(* IEC 61131-3 sources: teller/JD_Teller_LC2_V11/Class/CAIInputChannel, 1 file *)

(* ---- CAIInputChannel.st ---- *)
(*!
<Class
	Name               = "CAIInputChannel"
	Revision           = "2.20"
	RealtimeTask       = "false"
	CyclicTask         = "false"
	BackgroundTask     = "false"
	Sigmatek           = "true"
	OSInterface        = "false"
	HighPriority       = "false"
	Automatic          = "false"
	UpdateMode         = "Prescan"
	IconPath           = ".\Class\Tool.ico"
	SharedCommandTable = "true"
	Objectsize         = "(284,120)">
	<Channels>
		<Client Name="connectc" Required="true" Internal="false"/>
		<Client Name="EEOffset" Required="true" Internal="false"/>
		<Client Name="Neg" Required="false" Internal="false"/>
	</Channels>
	<RevDoku>
		<Owner Company="Sigmatek" Author="stewer"/>
		<Dokumentation Revision="2.20" Date="05.12.2013" Author="LanSte&#13;&#10;FucHer" Company="Sigmatek" Description="Added payload support&#13;&#10;Changed AWL code to Structured Text. CyRt Client default value: 1"/>
		<Dokumentation Revision="2.11" Date="04.03.2010" Author="BleErn" Company="Sigmatek" Description="Changes in BaseClass (UpdateRtPostScan)"/>
	</RevDoku>
	<Network Name="CAIInputChannel">
		<!-- List of Components in this network -->
		<Components>
			<Object
				Name       = "_base"
				Class      = "DAIInputChnl"
				Position   = "(270,150)"
				Visualized = "true">
				<Channels>
					<Server Name="Data"/>
					<Server Name="State"/>
					<Client Name="BitResolution"/>
					<Client Name="CBias"/>
					<Client Name="channel"/>
					<Client Name="CInvert"/>
					<Client Name="connect"/>
					<Client Name="CScale"/>
					<Client Name="CyRt" Value="1"/>
					<Client Name="TypeofChannel"/>
				</Channels>
			</Object>
		</Components>
		<Comments>
		</Comments>
		<!-- List of Connections in this network -->
		<Connections>
			<Connection Source="this.Data" Destination="_base.Data" Vertices="(742,210),(570,240),"/>
			<Connection Source="this.State" Destination="_base.State" Vertices="(742,270),(570,300),"/>
			<Connection Source="_base.TypeofChannel" Destination="this.TypeofChannel" Vertices="(270,360),(38,270),"/>
			<Connection Source="_base.CyRt" Destination="this.CyRt" Vertices="(270,420),(38,330),"/>
			<Connection Source="_base.CScale" Destination="this.CScale" Vertices="(270,480),(38,390),"/>
			<Connection Source="_base.CBias" Destination="this.CBias" Vertices="(270,540),(38,450),"/>
			<Connection Source="_base.CInvert" Destination="this.CInvert" Vertices="(270,600),(38,510),"/>
			<Connection Source="_base.BitResolution" Destination="this.BitResolution" Vertices="(270,660),(38,570),"/>
			<Connection Source="_base.channel" Destination="this.channel" Vertices="(270,240),(38,210),"/>
		</Connections>
		<!-- Headerfiles -->
		<Options>
		</Options>
	</Network>
</Class>
*)
#pragma using DAIInputChnl

CAIInputChannel : CLASS
: DAIInputChnl
  //Servers:
  //Clients:
	connectc 	: CltChCmd_HwBaseCDIAS;
	Neg 	: CltCh_DINT;
	EEOffset 	: CltCh_DINT;
  //Variables:
  //Functions:
				//! <Function Comment="[#ENGLISH]&#13;&#10; *******************************************************&#13;&#10; this is the init method of one input channel&#13;&#10; *******************************************************&#13;&#10;" Name="Init"/>
	FUNCTION VIRTUAL GLOBAL Init;

	FUNCTION CalFactory1;
				//! <Function Comment="-- overwite this function if there are other offsets ---------------------------&#13;&#10;" Name="GetEEOffset"/>
	FUNCTION VIRTUAL GLOBAL GetEEOffset
		VAR_OUTPUT
			Offset 	: UINT;
		END_VAR;

	FUNCTION GLOBAL ReCallFactory;

	FUNCTION VIRTUAL GLOBAL SetBalanceData;

	FUNCTION AWL CalFactory1_AWL;
  //Tables:
	FUNCTION @STD
		VAR_OUTPUT
			ret_code	: CONFSTATES;
		END_VAR;
	FUNCTION GLOBAL TAB @CT_;
END_CLASS;

#pragma usingLtd HwBaseCDIAS

#pragma usingLtd DiasMaster

(****************************************************************************************
*
*	Created : Sigmatek
*	Changes :
*		2.5 => 2.10	/	05.12.2007	/	Mark:	//#SR001
*			- [DB 713]: make compatible to CIV/DIV DataMover
*		1.1 => 2.5	/	06.03.2007	/	Mark:	//#SR000
*			- [DB 421]: now class is ready for plug & play over CIV
*		0.1 => 1.1 / 23.12.2004 / no Mark / ws
*			compatibility with Lasal Class 2
*			removed visible flags from internal servers
*
*****************************************************************************************)

//[#ENGLISH]
// *******************************************************
// this is the init method of one input channel
// *******************************************************
FUNCTION VIRTUAL GLOBAL CAIInputChannel::Init

	channel       := channel.read();
	TypeofChannel := TypeofChannel.read();
	CyRt          := CyRt.read();
	CScale        := CScale.read();
	CBias         := CBias.read();
	CInvert 	  := CInvert.read();
	BitResolution := BitResolution.read();
	Neg := Neg.Read();
	EEOffset := EEOffset.Read();

	if BitResolution = 14 then
		udMaxBin := 16000;
	else
		udMaxBin := 4000;
	end_if;

	//#SR000 start
	b_VaranAvailable := Connectc.Masterconnect.IsVaranAvailable() <> 0;

	if ( b_VaranAvailable = TRUE ) then
		if firstscan = 0 then
//#SR001			HandleRDValue:=connectc.AddOneChannel(thisp:=this, RTCY:=cyrt, channel:=channel);
			firstscan := 1;
		end_if;
	else
	//#SR000 end
		if connectc.GetEEState() then
			// no data on the EEPROM channel or wrong
			factory.dOffEE := 0;
			factory.dMulEE := 4000;
			factory.dDivEE := 4050;
			CalFactory1();
			if BitResolution = 14 then
				udMaxBin := 16383;
			else
				udMaxBin := 4095;
			end_if;
		else
			if firstscan = 0 then
				firstscan:=1;
				SetBalanceData();
				CalFactory1();
				HandleRDValue:=connectc.AddOneChannel(thisp:=this, RTCY:=cyrt, channel:=channel);
				if BitResolution = 14 then
					udMaxBin := 16383;
				else
					udMaxBin := 4095;
				end_if;
			end_if;
		end_if;
	end_if;		//#SR000

END_FUNCTION //VIRTUAL GLOBAL CAIInputChannel::Init
FUNCTION CAIInputChannel::CalFactory1

// -- calculate binary offset

  udBiasBin := (udMaxBin$DINT * CBias / -1000)$UDINT;
  udOffAct  := (udBiasBin$DINT * Factory.dDivEE / Factory.dMulEE + Factory.dOffEE)$UDINT;

// dMulAct

  if Neg = 0 then
    udMulAct := CScale$UDINT;
  else
    udMulAct := (CScale SHL 1)$UDINT;   // *2 weil +/-
  end_if;

// dDivAct

  udDivAct := ((udMaxBin + udBiasBin)$DINT * Factory.dDivEE / Factory.dMulEE)$UDINT;

END_FUNCTION // CAIInputChannel::CalFactory1
FUNCTION AWL CAIInputChannel::CalFactory1_AWL
#ifdef _LSL_TARGETARCH_X86
// -- calculate binary offset

         L.EAX     udMaxBin
         IMUL.D    cBias
         L.EBX     -1000
         IDIV      EBX
         S.EAX     udBiasBin

         IMUL.D    Factory.dDivEE
         IDIV.D    Factory.dMulEE
         ADD.EAX   Factory.dOffEE
         S.EAX     udOffAct

// dMulAct

         L.EAX     cScale
		 CMP.D	   Neg,0
		 JE		   noPlusMinus
		 SHL.EAX   1 // *2 weil +/-
noPlusMinus
         S.EAX     udMulAct

// dDivAct

         L.EAX     udMaxBin
         ADD.EAX   udBiasBin
         IMUL.D    Factory.dDivEE
         IDIV.D    Factory.dMulEE
         S.EAX     udDivAct
#endif
END_FUNCTION // CAIInputChannel::CalFactory1
//-- overwite this function if there are other offsets ---------------------------
FUNCTION VIRTUAL GLOBAL CAIInputChannel::GetEEOffset
VAR_OUTPUT
	Offset		: UINT;
END_VAR

	Offset := EEOffset$UINT + Channel$UINT * 6;

END_FUNCTION //VIRTUAL GLOBAL CAIInputChannel::GetEEOffset

FUNCTION GLOBAL CAIInputChannel::ReCallFactory			//#SR000

	if BitResolution = 14 then
		udMaxBin := 16000;
	else
		udMaxBin := 4000;
	end_if;

  SetBalanceData();

	CalFactory1();

	if BitResolution = 14 then
		udMaxBin := 16383;
	else
		udMaxBin := 4095;
	end_if;

	HandleRDValue:=connectc.AddOneChannel(thisp:=this, RTCY:=cyrt, channel:=channel);		//#SR001

END_FUNCTION //GLOBAL CAIInputChannel::ReCallFactory

FUNCTION VIRTUAL GLOBAL CAIInputChannel::SetBalanceData

  factory.dOffEE := TO_DINT (TO_INT(connectc.GetEEData(GetEEOffset()+0)));
  factory.dMulEE := TO_DINT (TO_INT(connectc.GetEEData(GetEEOffset()+2)));
  factory.dDivEE := TO_DINT (TO_INT(connectc.GetEEData(GetEEOffset()+4)));

  if factory.dMulEE = 0 |
     factory.dDivEE = 0 then

    factory.dMulEE := 4000;
    factory.dDivEE := 4050;

  end_if;

END_FUNCTION
